// TIA Portal V18 export
DATA_BLOCK "Functions"   // DB40
{ S7_Optimized_Access := 'TRUE' }
VERSION : 0.1
// stored: AutoNumber true, DBAccessibleFromOPCUA true, IsOnlyStoredInLoadMemory false, IsRetainMemResEnabled false, IsWriteProtectedInAS false, MemoryReserve 100
   VAR
      "Dosing function selected" : Bool;
      "Dosing Running" : Bool;
      "Dosing Completed" : Bool;
      "Function running" : Bool;
      "Esc Dosing function" : Bool;
      "Part present R Signal" : Bool;
      "start dosing by partpresent sensor" : Bool;
      "Start Dosing function" : Bool;
      "Start Dosing function site" : Bool;
      "Start dosing function HMI" : Bool;
      "Stop Dosing AB function" : Bool;
      "Stop Dosing B function" : Bool;
      "Stop Dosing A function" : Bool;
      "1k" : Struct
         "deaering A with valve selected" : Bool;
         "deaering B with valve  selected" : Bool;
         "deaering A without valve selected" : Bool;
         "deaering B without valve  selected" : Bool;
         "Flush selected" : Bool;
         "Flush selected during potlife" : Bool;
         "Condition Check A" : Bool;
         "Condition Check B" : Bool;
      END_STRUCT;
      "flush selection" : Struct
         "Flush A selected" : Bool;
         "Flush B selected" : Bool;
         "flush selection in HMI" : Bool;
      END_STRUCT;
      "2k" : Struct
         "metering program selected" : Bool;
         "pre run program selected" : Bool;
         "mixing ratio program selected" : Bool;
         "continous metering program selected" : Bool;
         "shot metering program selected" : Bool;
         "regeration program selected" : Bool;
      END_STRUCT;
      "Block all 1k metering" : Bool;
      "Block all 2k metering" : Bool;
      "Deselect all function" : Bool;
      "recirculation Selected" : Bool;
      "Pressure release selected" : Bool;
      "recirculation A selected" : Bool;
      "recirculation B selected" : Bool;
      "Pressure release A selected" : Bool;
      "Pressure release B selected" : Bool;
      "Stop Dosing function" : Bool;
      "stop dosing function site" : Bool;
      Functions : Int;
   END_VAR
   VAR RETAIN
      Auto : Bool;
   END_VAR
BEGIN
END_DATA_BLOCK
